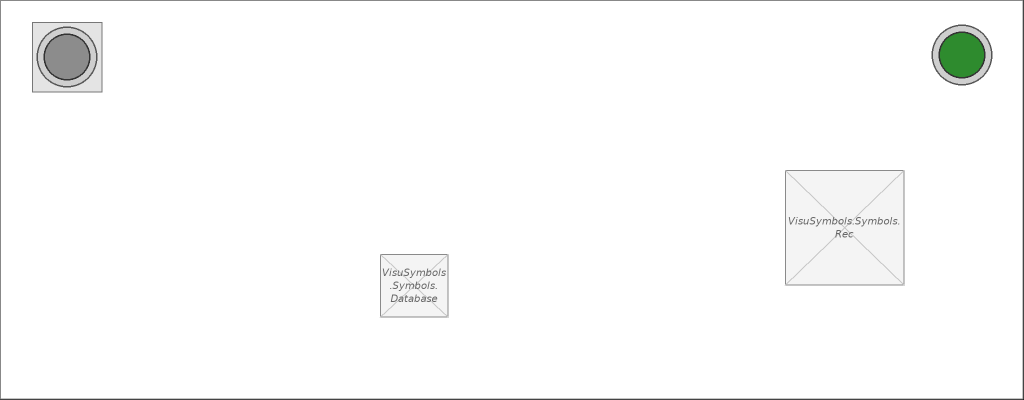
VISUALIZATION Startpage  // 1024x400
    RoundedRectangle (0,0 1024x400)
    PushSwitchLed (32,22 70x70), behaviour: TOGGLE, style: Switch-PushSwitchLed-Gray
    Lamp1 (927,20 70x70), style: Lamp-Lamp1-Green
    Image (785,170 119x115), image: VisuSymbols.Symbols.Rec
    Image (380,254 68x63), image: VisuSymbols.Symbols.Database
END_VISUALIZATION

(* stored: Version 1.1.0.1, ProductVersion 3.1.4024.12
   Visu Startpage: Id {17b444b5-9ab4-4887-acae-4769a5819030} *)
